(*
Integrates the input error signal over time.

The output accumulates the input scaled by the integral gain :math:`K_i = 1 / T_n`,
and is clamped to [:attr:`Minimum`, :attr:`Maximum`] on every cycle.
Setting :attr:`Tn` to ``LTIME#0`` disables integration, setting the output to zero.

Use :meth:`Sync` to preset the integrator state for bumpless transfer when
switching from manual to automatic mode.

.. note::
   Set :attr:`Maximum` before :attr:`Minimum` to ensure the clamp guard applies
   correctly.

   Use ``FB_init`` to set :attr:`tTn` at declaration time.
*)
{attribute 'no_assign'}
{attribute 'enable_dynamic_creation'}
{attribute 'no_explicit_call' := 'direct call for this function block is not allowed'}
FUNCTION_BLOCK FB_Integrator EXTENDS FB_SisoComponent
IMPLEMENTS FsCommon.I_Runnable, I_Resettable, I_Bounded
VAR
	_tTn   		: LTIME; // Integral action time (Tn).
	_bSync 		: BOOL;  // Triggers a bumpless transfer on the next Run call.
	_fSync 		: LREAL; // Target integrator state for bumpless transfer.
	_fMaximum   : LREAL := FsCommon.GVL_TypeValueLimits.LREAL_MAX; // Upper output clamp. Clamped to >= Minimum.
	_fMinimum   : LREAL := FsCommon.GVL_TypeValueLimits.LREAL_MIN; // Lower output clamp. Clamped to <= Maximum.
END_VAR

METHOD FB_init : BOOL
VAR_INPUT
	bInitRetains : BOOL;  // if TRUE, the retain variables are initialized (warm start / cold start)
	bInCopyCode  : BOOL;  // if TRUE, the instance afterwards gets moved into the copy code (online change)
	tTn          : LTIME; // Integral action time. LTIME#0 disables integration.
END_VAR
THIS^._tTn := tTn;
END_METHOD

(*
Gets or sets the upper output clamp.

Internally clamped to be greater than or equal to :attr:`Minimum`.
Set this before :attr:`Minimum` to ensure the guard applies correctly.
*)
PROPERTY Maximum : LREAL
GET
Maximum := THIS^._fMaximum;
END_GET
SET
THIS^._fMaximum := MAX(THIS^._fMinimum, Maximum);
END_SET
END_PROPERTY

(*
Gets or sets the lower output clamp.

Internally clamped to be less than or equal to :attr:`Maximum`.
Set :attr:`Maximum` before this property to ensure the guard applies correctly.
*)
PROPERTY Minimum : LREAL
GET
Minimum := THIS^._fMinimum;
END_GET
SET
THIS^._fMinimum := MIN(THIS^._fMaximum, Minimum);
END_SET
END_PROPERTY

(* Clears the integrator state and output. *)
METHOD Reset
VAR_INPUT
END_VAR
THIS^._fOutput := 0;
END_METHOD

(*
Advances the integrator by one time step.

.. note::
   Must be called once per cycle on a single PLC task. If :attr:`Tn` is
   ``LTIME#0`` the output is set to zero.
*)
METHOD Run
VAR_INST
	{attribute 'hide'}
	bInit       : BOOL := TRUE;
	{attribute 'hide'}
	fT          : LREAL;
	{attribute 'hide'}
	fbTaskCycle : FsCommon.FB_PlcTaskCycleChangeDetector(0);
END_VAR
IF bInit THEN
	fT := TO_LREAL(FsCommon.F_GetCurrentTaskCycleTime()) / TO_LREAL(LTIME#1S);
	RETURN(bInit := fT <= 0);
	fbTaskCycle.TaskIndex := FsCommon.F_GetCurrentTaskIndex();
END_IF

RETURN(NOT fbTaskCycle.HasChanged);

THIS^._fMaximum := MAX(THIS^._fMinimum, THIS^._fMaximum);
THIS^._fMinimum := MIN(THIS^._fMinimum, THIS^._fMaximum);

IF FsCommon.F_ResetOnTrue(THIS^._bSync) THEN
	THIS^._fOutput := THIS^._fSync;
END_IF

IF THIS^._tTn = LTIME#0S THEN
	THIS^._fOutput := 0;
	RETURN;
END_IF

THIS^._fOutput := LIMIT(
	THIS^._fMinimum, 
	THIS^._fOutput + 
		(1.0 / (TO_LREAL(THIS^._tTn) / TO_LREAL(LTIME#1S))) * THIS^._fInput * fT,
	THIS^._fMaximum
);
END_METHOD

(*
Forces the integrator state to a given value on the next :meth:`Run` call.

Use this for bumpless transfer when switching from manual to automatic mode,
to prevent a sudden jump in output.
*)
METHOD Sync
VAR_INPUT
	// Target integrator state.
	fValue : LREAL; 
END_VAR
THIS^._bSync := TRUE;
THIS^._fSync := fValue;
END_METHOD

(*
Gets or sets the integral action time (Tn).

This controls how aggressively the integrator responds to sustained error.
A shorter value increases integral action. Setting it to ``LTIME#0`` disables
integration entirely, setting the output to zero.
*)
PROPERTY Tn : LTIME
GET
Tn := THIS^._tTn;
END_GET
SET
THIS^._tTn := Tn;
END_SET
END_PROPERTY

END_FUNCTION_BLOCK

(* stored: Version 1.1.0.1, ProductVersion 3.1.4024.15
   POU FB_Integrator: Id {7ca0c08c-f207-4eb5-a0d9-54bd93c65f82}, SpecialFunc None
   Method FB_init: Id {c6dade2a-2d12-4771-892f-f8afbd0a6039}
   Property Maximum: Id {b7589c00-7ee0-4541-93bc-2e57fc1f93bc}
   Get Get: Id {983b9dbc-0394-452d-bab5-7875c0d74c9b}
   Set Set: Id {608c7a5d-ebf1-4e44-8ba6-ce7a9f38c421}
   Property Minimum: Id {fc41bd10-44e9-4e18-8de2-b1ec342a3857}
   Get Get: Id {c60fdb29-7826-4aae-ac55-ecaabda6d860}
   Set Set: Id {43bfea17-b59b-49cd-8d17-5fa230e5164e}
   Method Reset: Id {063453a7-8d9c-4532-8c8c-9af5dcadd63c}
   Method Run: Id {ba620ebb-bf63-48bd-b3f8-0aba28bc3078}
   Method Sync: Id {0664633e-4340-481c-9446-e6a9c9436467}
   Property Tn: Id {61d77439-5454-4fcc-b881-c1903dc5075a}
   Get Get: Id {c3ffca41-92c7-4f88-af72-22b19b0f5702}
   Set Set: Id {1f4b5be9-6245-47b7-ba3e-e6c4ef0a1dba} *)
